! Draw black
MoveJ Offs(Target_drawing_origin,0,0,0),v100,fine,PencilHolder\WObj:=PAPER;
MoveL Offs(Target_drawing_origin,0,0,0),v50,fine,PencilHolder\WObj:=PAPER;
MoveL Offs(Target_drawing_origin,-53,0,0),v50,fine,PencilHolder\WObj:=PAPER;
MoveL Offs(Target_drawing_origin,0,1,0),v50,fine,PencilHolder\WObj:=PAPER;
MoveL Offs(Target_drawing_origin,-53,1,0),v50,fine,PencilHolder\WObj:=PAPER;
MoveL Offs(Target_drawing_origin,0,2,0),v50,fine,PencilHolder\WObj:=PAPER;
MoveL Offs(Target_drawing_origin,-53,2,0),v50,fine,PencilHolder\WObj:=PAPER;
MoveL Offs(Target_drawing_origin,0,3,0),v50,fine,PencilHolder\WObj:=PAPER;
MoveL Offs(Target_drawing_origin,-53,3,0),v50,fine,PencilHolder\WObj:=PAPER;
MoveL Offs(Target_drawing_origin,0,4,0),v50,fine,PencilHolder\WObj:=PAPER;
MoveL Offs(Target_drawing_origin,-53,4,0),v50,fine,PencilHolder\WObj:=PAPER;
MoveL Offs(Target_drawing_origin,0,5,0),v50,fine,PencilHolder\WObj:=PAPER;
MoveL Offs(Target_drawing_origin,-53,5,0),v50,fine,PencilHolder\WObj:=PAPER;
MoveL Offs(Target_drawing_origin,0,6,0),v50,fine,PencilHolder\WObj:=PAPER;
MoveL Offs(Target_drawing_origin,-58,6,0),v50,fine,PencilHolder\WObj:=PAPER;
MoveL Offs(Target_drawing_origin,0,7,0),v50,fine,PencilHolder\WObj:=PAPER;
MoveL Offs(Target_drawing_origin,-58,7,0),v50,fine,PencilHolder\WObj:=PAPER;
MoveL Offs(Target_drawing_origin,0,8,0),v50,fine,PencilHolder\WObj:=PAPER;
MoveL Offs(Target_drawing_origin,-58,8,0),v50,fine,PencilHolder\WObj:=PAPER;
MoveL Offs(Target_drawing_origin,0,9,0),v50,fine,PencilHolder\WObj:=PAPER;
MoveL Offs(Target_drawing_origin,-58,9,0),v50,fine,PencilHolder\WObj:=PAPER;
MoveL Offs(Target_drawing_origin,0,10,0),v50,fine,PencilHolder\WObj:=PAPER;
MoveL Offs(Target_drawing_origin,-58,10,0),v50,fine,PencilHolder\WObj:=PAPER;
MoveL Offs(Target_drawing_origin,0,11,0),v50,fine,PencilHolder\WObj:=PAPER;
MoveL Offs(Target_drawing_origin,-58,11,0),v50,fine,PencilHolder\WObj:=PAPER;
MoveL Offs(Target_drawing_origin,0,12,0),v50,fine,PencilHolder\WObj:=PAPER;
MoveL Offs(Target_drawing_origin,-58,12,0),v50,fine,PencilHolder\WObj:=PAPER;
MoveL Offs(Target_drawing_origin,0,13,0),v50,fine,PencilHolder\WObj:=PAPER;
MoveL Offs(Target_drawing_origin,-58,13,0),v50,fine,PencilHolder\WObj:=PAPER;
MoveL Offs(Target_drawing_origin,0,14,0),v50,fine,PencilHolder\WObj:=PAPER;
MoveL Offs(Target_drawing_origin,-58,14,0),v50,fine,PencilHolder\WObj:=PAPER;
MoveL Offs(Target_drawing_origin,0,15,0),v50,fine,PencilHolder\WObj:=PAPER;
MoveL Offs(Target_drawing_origin,-58,15,0),v50,fine,PencilHolder\WObj:=PAPER;
MoveL Offs(Target_drawing_origin,0,16,0),v50,fine,PencilHolder\WObj:=PAPER;
MoveL Offs(Target_drawing_origin,-15,16,0),v50,fine,PencilHolder\WObj:=PAPER;
MoveL Offs(Target_drawing_origin,-27,16,0),v50,fine,PencilHolder\WObj:=PAPER;
MoveL Offs(Target_drawing_origin,-58,16,0),v50,fine,PencilHolder\WObj:=PAPER;
MoveL Offs(Target_drawing_origin,0,17,0),v50,fine,PencilHolder\WObj:=PAPER;
MoveL Offs(Target_drawing_origin,-15,17,0),v50,fine,PencilHolder\WObj:=PAPER;
MoveL Offs(Target_drawing_origin,-27,17,0),v50,fine,PencilHolder\WObj:=PAPER;
MoveL Offs(Target_drawing_origin,-58,17,0),v50,fine,PencilHolder\WObj:=PAPER;
MoveL Offs(Target_drawing_origin,0,18,0),v50,fine,PencilHolder\WObj:=PAPER;
MoveL Offs(Target_drawing_origin,-15,18,0),v50,fine,PencilHolder\WObj:=PAPER;
MoveL Offs(Target_drawing_origin,-27,18,0),v50,fine,PencilHolder\WObj:=PAPER;
MoveL Offs(Target_drawing_origin,-58,18,0),v50,fine,PencilHolder\WObj:=PAPER;
MoveL Offs(Target_drawing_origin,0,19,0),v50,fine,PencilHolder\WObj:=PAPER;
MoveL Offs(Target_drawing_origin,-15,19,0),v50,fine,PencilHolder\WObj:=PAPER;
MoveL Offs(Target_drawing_origin,-27,19,0),v50,fine,PencilHolder\WObj:=PAPER;
MoveL Offs(Target_drawing_origin,-58,19,0),v50,fine,PencilHolder\WObj:=PAPER;
MoveL Offs(Target_drawing_origin,0,20,0),v50,fine,PencilHolder\WObj:=PAPER;
MoveL Offs(Target_drawing_origin,-15,20,0),v50,fine,PencilHolder\WObj:=PAPER;
MoveL Offs(Target_drawing_origin,-27,20,0),v50,fine,PencilHolder\WObj:=PAPER;
MoveL Offs(Target_drawing_origin,-58,20,0),v50,fine,PencilHolder\WObj:=PAPER;
MoveL Offs(Target_drawing_origin,-27,21,0),v50,fine,PencilHolder\WObj:=PAPER;
MoveL Offs(Target_drawing_origin,-58,21,0),v50,fine,PencilHolder\WObj:=PAPER;
MoveL Offs(Target_drawing_origin,-27,22,0),v50,fine,PencilHolder\WObj:=PAPER;
MoveL Offs(Target_drawing_origin,-58,22,0),v50,fine,PencilHolder\WObj:=PAPER;
MoveL Offs(Target_drawing_origin,-27,23,0),v50,fine,PencilHolder\WObj:=PAPER;
MoveL Offs(Target_drawing_origin,-58,23,0),v50,fine,PencilHolder\WObj:=PAPER;
MoveL Offs(Target_drawing_origin,-27,24,0),v50,fine,PencilHolder\WObj:=PAPER;
MoveL Offs(Target_drawing_origin,-58,24,0),v50,fine,PencilHolder\WObj:=PAPER;
MoveL Offs(Target_drawing_origin,-27,25,0),v50,fine,PencilHolder\WObj:=PAPER;
MoveL Offs(Target_drawing_origin,-58,25,0),v50,fine,PencilHolder\WObj:=PAPER;
MoveL Offs(Target_drawing_origin,-27,26,0),v50,fine,PencilHolder\WObj:=PAPER;
MoveL Offs(Target_drawing_origin,-58,26,0),v50,fine,PencilHolder\WObj:=PAPER;
MoveL Offs(Target_drawing_origin,-17,27,0),v50,fine,PencilHolder\WObj:=PAPER;
MoveL Offs(Target_drawing_origin,-58,27,0),v50,fine,PencilHolder\WObj:=PAPER;
MoveL Offs(Target_drawing_origin,-16,28,0),v50,fine,PencilHolder\WObj:=PAPER;
MoveL Offs(Target_drawing_origin,-58,28,0),v50,fine,PencilHolder\WObj:=PAPER;
MoveL Offs(Target_drawing_origin,-16,29,0),v50,fine,PencilHolder\WObj:=PAPER;
MoveL Offs(Target_drawing_origin,-58,29,0),v50,fine,PencilHolder\WObj:=PAPER;
MoveL Offs(Target_drawing_origin,-16,30,0),v50,fine,PencilHolder\WObj:=PAPER;
MoveL Offs(Target_drawing_origin,-58,30,0),v50,fine,PencilHolder\WObj:=PAPER;
MoveL Offs(Target_drawing_origin,-16,31,0),v50,fine,PencilHolder\WObj:=PAPER;
MoveL Offs(Target_drawing_origin,-58,31,0),v50,fine,PencilHolder\WObj:=PAPER;
MoveL Offs(Target_drawing_origin,-16,32,0),v50,fine,PencilHolder\WObj:=PAPER;
MoveL Offs(Target_drawing_origin,-58,32,0),v50,fine,PencilHolder\WObj:=PAPER;
MoveL Offs(Target_drawing_origin,-16,33,0),v50,fine,PencilHolder\WObj:=PAPER;
MoveL Offs(Target_drawing_origin,-58,33,0),v50,fine,PencilHolder\WObj:=PAPER;
MoveL Offs(Target_drawing_origin,-16,34,0),v50,fine,PencilHolder\WObj:=PAPER;
MoveL Offs(Target_drawing_origin,-58,34,0),v50,fine,PencilHolder\WObj:=PAPER;
MoveL Offs(Target_drawing_origin,-16,35,0),v50,fine,PencilHolder\WObj:=PAPER;
MoveL Offs(Target_drawing_origin,-58,35,0),v50,fine,PencilHolder\WObj:=PAPER;
MoveL Offs(Target_drawing_origin,-16,36,0),v50,fine,PencilHolder\WObj:=PAPER;
MoveL Offs(Target_drawing_origin,-58,36,0),v50,fine,PencilHolder\WObj:=PAPER;
MoveL Offs(Target_drawing_origin,-16,37,0),v50,fine,PencilHolder\WObj:=PAPER;
MoveL Offs(Target_drawing_origin,-58,37,0),v50,fine,PencilHolder\WObj:=PAPER;
MoveL Offs(Target_drawing_origin,-11,38,0),v50,fine,PencilHolder\WObj:=PAPER;
MoveL Offs(Target_drawing_origin,-53,38,0),v50,fine,PencilHolder\WObj:=PAPER;
MoveL Offs(Target_drawing_origin,-11,39,0),v50,fine,PencilHolder\WObj:=PAPER;
MoveL Offs(Target_drawing_origin,-53,39,0),v50,fine,PencilHolder\WObj:=PAPER;
MoveL Offs(Target_drawing_origin,-11,40,0),v50,fine,PencilHolder\WObj:=PAPER;
MoveL Offs(Target_drawing_origin,-53,40,0),v50,fine,PencilHolder\WObj:=PAPER;
MoveL Offs(Target_drawing_origin,-11,41,0),v50,fine,PencilHolder\WObj:=PAPER;
MoveL Offs(Target_drawing_origin,-53,41,0),v50,fine,PencilHolder\WObj:=PAPER;
MoveL Offs(Target_drawing_origin,-11,42,0),v50,fine,PencilHolder\WObj:=PAPER;
MoveL Offs(Target_drawing_origin,-53,42,0),v50,fine,PencilHolder\WObj:=PAPER;
MoveL Offs(Target_drawing_origin,-11,43,0),v50,fine,PencilHolder\WObj:=PAPER;
MoveL Offs(Target_drawing_origin,-42,43,0),v50,fine,PencilHolder\WObj:=PAPER;
MoveL Offs(Target_drawing_origin,-6,44,0),v50,fine,PencilHolder\WObj:=PAPER;
MoveL Offs(Target_drawing_origin,-42,44,0),v50,fine,PencilHolder\WObj:=PAPER;
MoveL Offs(Target_drawing_origin,-76,44,0),v50,fine,PencilHolder\WObj:=PAPER;
MoveL Offs(Target_drawing_origin,-96,44,0),v50,fine,PencilHolder\WObj:=PAPER;
MoveL Offs(Target_drawing_origin,-6,45,0),v50,fine,PencilHolder\WObj:=PAPER;
MoveL Offs(Target_drawing_origin,-42,45,0),v50,fine,PencilHolder\WObj:=PAPER;
MoveL Offs(Target_drawing_origin,-76,45,0),v50,fine,PencilHolder\WObj:=PAPER;
MoveL Offs(Target_drawing_origin,-96,45,0),v50,fine,PencilHolder\WObj:=PAPER;
MoveL Offs(Target_drawing_origin,-6,46,0),v50,fine,PencilHolder\WObj:=PAPER;
MoveL Offs(Target_drawing_origin,-42,46,0),v50,fine,PencilHolder\WObj:=PAPER;
MoveL Offs(Target_drawing_origin,-76,46,0),v50,fine,PencilHolder\WObj:=PAPER;
MoveL Offs(Target_drawing_origin,-96,46,0),v50,fine,PencilHolder\WObj:=PAPER;
MoveL Offs(Target_drawing_origin,-6,47,0),v50,fine,PencilHolder\WObj:=PAPER;
MoveL Offs(Target_drawing_origin,-42,47,0),v50,fine,PencilHolder\WObj:=PAPER;
MoveL Offs(Target_drawing_origin,-76,47,0),v50,fine,PencilHolder\WObj:=PAPER;
MoveL Offs(Target_drawing_origin,-96,47,0),v50,fine,PencilHolder\WObj:=PAPER;
MoveL Offs(Target_drawing_origin,-6,48,0),v50,fine,PencilHolder\WObj:=PAPER;
MoveL Offs(Target_drawing_origin,-37,48,0),v50,fine,PencilHolder\WObj:=PAPER;
MoveL Offs(Target_drawing_origin,-76,48,0),v50,fine,PencilHolder\WObj:=PAPER;
MoveL Offs(Target_drawing_origin,-96,48,0),v50,fine,PencilHolder\WObj:=PAPER;
MoveL Offs(Target_drawing_origin,0,49,0),v50,fine,PencilHolder\WObj:=PAPER;
MoveL Offs(Target_drawing_origin,-37,49,0),v50,fine,PencilHolder\WObj:=PAPER;
MoveL Offs(Target_drawing_origin,-71,49,0),v50,fine,PencilHolder\WObj:=PAPER;
MoveL Offs(Target_drawing_origin,-101,49,0),v50,fine,PencilHolder\WObj:=PAPER;
MoveL Offs(Target_drawing_origin,0,50,0),v50,fine,PencilHolder\WObj:=PAPER;
MoveL Offs(Target_drawing_origin,-37,50,0),v50,fine,PencilHolder\WObj:=PAPER;
MoveL Offs(Target_drawing_origin,-71,50,0),v50,fine,PencilHolder\WObj:=PAPER;
MoveL Offs(Target_drawing_origin,-101,50,0),v50,fine,PencilHolder\WObj:=PAPER;
MoveL Offs(Target_drawing_origin,0,51,0),v50,fine,PencilHolder\WObj:=PAPER;
MoveL Offs(Target_drawing_origin,-37,51,0),v50,fine,PencilHolder\WObj:=PAPER;
MoveL Offs(Target_drawing_origin,-71,51,0),v50,fine,PencilHolder\WObj:=PAPER;
MoveL Offs(Target_drawing_origin,-101,51,0),v50,fine,PencilHolder\WObj:=PAPER;
MoveL Offs(Target_drawing_origin,0,52,0),v50,fine,PencilHolder\WObj:=PAPER;
MoveL Offs(Target_drawing_origin,-37,52,0),v50,fine,PencilHolder\WObj:=PAPER;
MoveL Offs(Target_drawing_origin,-71,52,0),v50,fine,PencilHolder\WObj:=PAPER;
MoveL Offs(Target_drawing_origin,-101,52,0),v50,fine,PencilHolder\WObj:=PAPER;
MoveL Offs(Target_drawing_origin,0,53,0),v50,fine,PencilHolder\WObj:=PAPER;
MoveL Offs(Target_drawing_origin,-37,53,0),v50,fine,PencilHolder\WObj:=PAPER;
MoveL Offs(Target_drawing_origin,-71,53,0),v50,fine,PencilHolder\WObj:=PAPER;
MoveL Offs(Target_drawing_origin,-101,53,0),v50,fine,PencilHolder\WObj:=PAPER;
MoveL Offs(Target_drawing_origin,0,54,0),v50,fine,PencilHolder\WObj:=PAPER;
MoveL Offs(Target_drawing_origin,-31,54,0),v50,fine,PencilHolder\WObj:=PAPER;
MoveL Offs(Target_drawing_origin,-60,54,0),v50,fine,PencilHolder\WObj:=PAPER;
MoveL Offs(Target_drawing_origin,-107,54,0),v50,fine,PencilHolder\WObj:=PAPER;
MoveL Offs(Target_drawing_origin,0,55,0),v50,fine,PencilHolder\WObj:=PAPER;
MoveL Offs(Target_drawing_origin,-31,55,0),v50,fine,PencilHolder\WObj:=PAPER;
MoveL Offs(Target_drawing_origin,-60,55,0),v50,fine,PencilHolder\WObj:=PAPER;
MoveL Offs(Target_drawing_origin,-107,55,0),v50,fine,PencilHolder\WObj:=PAPER;
MoveL Offs(Target_drawing_origin,0,56,0),v50,fine,PencilHolder\WObj:=PAPER;
MoveL Offs(Target_drawing_origin,-31,56,0),v50,fine,PencilHolder\WObj:=PAPER;
MoveL Offs(Target_drawing_origin,-60,56,0),v50,fine,PencilHolder\WObj:=PAPER;
MoveL Offs(Target_drawing_origin,-107,56,0),v50,fine,PencilHolder\WObj:=PAPER;
MoveL Offs(Target_drawing_origin,0,57,0),v50,fine,PencilHolder\WObj:=PAPER;
MoveL Offs(Target_drawing_origin,-31,57,0),v50,fine,PencilHolder\WObj:=PAPER;
MoveL Offs(Target_drawing_origin,-60,57,0),v50,fine,PencilHolder\WObj:=PAPER;
MoveL Offs(Target_drawing_origin,-107,57,0),v50,fine,PencilHolder\WObj:=PAPER;
MoveL Offs(Target_drawing_origin,0,58,0),v50,fine,PencilHolder\WObj:=PAPER;
MoveL Offs(Target_drawing_origin,-31,58,0),v50,fine,PencilHolder\WObj:=PAPER;
MoveL Offs(Target_drawing_origin,-60,58,0),v50,fine,PencilHolder\WObj:=PAPER;
MoveL Offs(Target_drawing_origin,-107,58,0),v50,fine,PencilHolder\WObj:=PAPER;
MoveL Offs(Target_drawing_origin,0,59,0),v50,fine,PencilHolder\WObj:=PAPER;
MoveL Offs(Target_drawing_origin,-31,59,0),v50,fine,PencilHolder\WObj:=PAPER;
MoveL Offs(Target_drawing_origin,-60,59,0),v50,fine,PencilHolder\WObj:=PAPER;
MoveL Offs(Target_drawing_origin,-107,59,0),v50,fine,PencilHolder\WObj:=PAPER;
MoveL Offs(Target_drawing_origin,0,60,0),v50,fine,PencilHolder\WObj:=PAPER;
MoveL Offs(Target_drawing_origin,-112,60,0),v50,fine,PencilHolder\WObj:=PAPER;
MoveL Offs(Target_drawing_origin,0,61,0),v50,fine,PencilHolder\WObj:=PAPER;
MoveL Offs(Target_drawing_origin,-112,61,0),v50,fine,PencilHolder\WObj:=PAPER;
MoveL Offs(Target_drawing_origin,0,62,0),v50,fine,PencilHolder\WObj:=PAPER;
MoveL Offs(Target_drawing_origin,-112,62,0),v50,fine,PencilHolder\WObj:=PAPER;
MoveL Offs(Target_drawing_origin,0,63,0),v50,fine,PencilHolder\WObj:=PAPER;
MoveL Offs(Target_drawing_origin,-112,63,0),v50,fine,PencilHolder\WObj:=PAPER;
MoveL Offs(Target_drawing_origin,0,64,0),v50,fine,PencilHolder\WObj:=PAPER;
MoveL Offs(Target_drawing_origin,-112,64,0),v50,fine,PencilHolder\WObj:=PAPER;
MoveL Offs(Target_drawing_origin,0,65,0),v50,fine,PencilHolder\WObj:=PAPER;
MoveL Offs(Target_drawing_origin,-112,65,0),v50,fine,PencilHolder\WObj:=PAPER;
MoveL Offs(Target_drawing_origin,0,66,0),v50,fine,PencilHolder\WObj:=PAPER;
MoveL Offs(Target_drawing_origin,-118,66,0),v50,fine,PencilHolder\WObj:=PAPER;
MoveL Offs(Target_drawing_origin,0,67,0),v50,fine,PencilHolder\WObj:=PAPER;
MoveL Offs(Target_drawing_origin,-118,67,0),v50,fine,PencilHolder\WObj:=PAPER;
MoveL Offs(Target_drawing_origin,0,68,0),v50,fine,PencilHolder\WObj:=PAPER;
MoveL Offs(Target_drawing_origin,-118,68,0),v50,fine,PencilHolder\WObj:=PAPER;
MoveL Offs(Target_drawing_origin,0,69,0),v50,fine,PencilHolder\WObj:=PAPER;
MoveL Offs(Target_drawing_origin,-118,69,0),v50,fine,PencilHolder\WObj:=PAPER;
MoveL Offs(Target_drawing_origin,-5,70,0),v50,fine,PencilHolder\WObj:=PAPER;
MoveL Offs(Target_drawing_origin,-118,70,0),v50,fine,PencilHolder\WObj:=PAPER;
MoveL Offs(Target_drawing_origin,-6,71,0),v50,fine,PencilHolder\WObj:=PAPER;
MoveL Offs(Target_drawing_origin,-123,71,0),v50,fine,PencilHolder\WObj:=PAPER;
MoveL Offs(Target_drawing_origin,-6,72,0),v50,fine,PencilHolder\WObj:=PAPER;
MoveL Offs(Target_drawing_origin,-123,72,0),v50,fine,PencilHolder\WObj:=PAPER;
MoveL Offs(Target_drawing_origin,-6,73,0),v50,fine,PencilHolder\WObj:=PAPER;
MoveL Offs(Target_drawing_origin,-123,73,0),v50,fine,PencilHolder\WObj:=PAPER;
MoveL Offs(Target_drawing_origin,-6,74,0),v50,fine,PencilHolder\WObj:=PAPER;
MoveL Offs(Target_drawing_origin,-123,74,0),v50,fine,PencilHolder\WObj:=PAPER;
MoveL Offs(Target_drawing_origin,-6,75,0),v50,fine,PencilHolder\WObj:=PAPER;
MoveL Offs(Target_drawing_origin,-123,75,0),v50,fine,PencilHolder\WObj:=PAPER;
MoveL Offs(Target_drawing_origin,-11,76,0),v50,fine,PencilHolder\WObj:=PAPER;
MoveL Offs(Target_drawing_origin,-74,76,0),v50,fine,PencilHolder\WObj:=PAPER;
MoveL Offs(Target_drawing_origin,-92,76,0),v50,fine,PencilHolder\WObj:=PAPER;
MoveL Offs(Target_drawing_origin,-123,76,0),v50,fine,PencilHolder\WObj:=PAPER;
MoveL Offs(Target_drawing_origin,-11,77,0),v50,fine,PencilHolder\WObj:=PAPER;
MoveL Offs(Target_drawing_origin,-74,77,0),v50,fine,PencilHolder\WObj:=PAPER;
MoveL Offs(Target_drawing_origin,-92,77,0),v50,fine,PencilHolder\WObj:=PAPER;
MoveL Offs(Target_drawing_origin,-123,77,0),v50,fine,PencilHolder\WObj:=PAPER;
MoveL Offs(Target_drawing_origin,-11,78,0),v50,fine,PencilHolder\WObj:=PAPER;
MoveL Offs(Target_drawing_origin,-74,78,0),v50,fine,PencilHolder\WObj:=PAPER;
MoveL Offs(Target_drawing_origin,-92,78,0),v50,fine,PencilHolder\WObj:=PAPER;
MoveL Offs(Target_drawing_origin,-123,78,0),v50,fine,PencilHolder\WObj:=PAPER;
MoveL Offs(Target_drawing_origin,-11,79,0),v50,fine,PencilHolder\WObj:=PAPER;
MoveL Offs(Target_drawing_origin,-74,79,0),v50,fine,PencilHolder\WObj:=PAPER;
MoveL Offs(Target_drawing_origin,-92,79,0),v50,fine,PencilHolder\WObj:=PAPER;
MoveL Offs(Target_drawing_origin,-123,79,0),v50,fine,PencilHolder\WObj:=PAPER;
MoveL Offs(Target_drawing_origin,-11,80,0),v50,fine,PencilHolder\WObj:=PAPER;
MoveL Offs(Target_drawing_origin,-74,80,0),v50,fine,PencilHolder\WObj:=PAPER;
MoveL Offs(Target_drawing_origin,-92,80,0),v50,fine,PencilHolder\WObj:=PAPER;
MoveL Offs(Target_drawing_origin,-123,80,0),v50,fine,PencilHolder\WObj:=PAPER;
MoveL Offs(Target_drawing_origin,-16,81,0),v50,fine,PencilHolder\WObj:=PAPER;
MoveL Offs(Target_drawing_origin,-69,81,0),v50,fine,PencilHolder\WObj:=PAPER;
MoveL Offs(Target_drawing_origin,-92,81,0),v50,fine,PencilHolder\WObj:=PAPER;
MoveL Offs(Target_drawing_origin,-123,81,0),v50,fine,PencilHolder\WObj:=PAPER;
MoveL Offs(Target_drawing_origin,-16,82,0),v50,fine,PencilHolder\WObj:=PAPER;
MoveL Offs(Target_drawing_origin,-69,82,0),v50,fine,PencilHolder\WObj:=PAPER;
MoveL Offs(Target_drawing_origin,-92,82,0),v50,fine,PencilHolder\WObj:=PAPER;
MoveL Offs(Target_drawing_origin,-123,82,0),v50,fine,PencilHolder\WObj:=PAPER;
MoveL Offs(Target_drawing_origin,-16,83,0),v50,fine,PencilHolder\WObj:=PAPER;
MoveL Offs(Target_drawing_origin,-69,83,0),v50,fine,PencilHolder\WObj:=PAPER;
MoveL Offs(Target_drawing_origin,-92,83,0),v50,fine,PencilHolder\WObj:=PAPER;
MoveL Offs(Target_drawing_origin,-123,83,0),v50,fine,PencilHolder\WObj:=PAPER;
MoveL Offs(Target_drawing_origin,-16,84,0),v50,fine,PencilHolder\WObj:=PAPER;
MoveL Offs(Target_drawing_origin,-69,84,0),v50,fine,PencilHolder\WObj:=PAPER;
MoveL Offs(Target_drawing_origin,-92,84,0),v50,fine,PencilHolder\WObj:=PAPER;
MoveL Offs(Target_drawing_origin,-123,84,0),v50,fine,PencilHolder\WObj:=PAPER;
MoveL Offs(Target_drawing_origin,-16,85,0),v50,fine,PencilHolder\WObj:=PAPER;
MoveL Offs(Target_drawing_origin,-69,85,0),v50,fine,PencilHolder\WObj:=PAPER;
MoveL Offs(Target_drawing_origin,-92,85,0),v50,fine,PencilHolder\WObj:=PAPER;
MoveL Offs(Target_drawing_origin,-123,85,0),v50,fine,PencilHolder\WObj:=PAPER;
MoveL Offs(Target_drawing_origin,-21,86,0),v50,fine,PencilHolder\WObj:=PAPER;
MoveL Offs(Target_drawing_origin,-64,86,0),v50,fine,PencilHolder\WObj:=PAPER;
MoveL Offs(Target_drawing_origin,-92,86,0),v50,fine,PencilHolder\WObj:=PAPER;
MoveL Offs(Target_drawing_origin,-123,86,0),v50,fine,PencilHolder\WObj:=PAPER;
MoveL Offs(Target_drawing_origin,-22,87,0),v50,fine,PencilHolder\WObj:=PAPER;
MoveL Offs(Target_drawing_origin,-64,87,0),v50,fine,PencilHolder\WObj:=PAPER;
MoveL Offs(Target_drawing_origin,-87,87,0),v50,fine,PencilHolder\WObj:=PAPER;
MoveL Offs(Target_drawing_origin,-123,87,0),v50,fine,PencilHolder\WObj:=PAPER;
MoveL Offs(Target_drawing_origin,-22,88,0),v50,fine,PencilHolder\WObj:=PAPER;
MoveL Offs(Target_drawing_origin,-64,88,0),v50,fine,PencilHolder\WObj:=PAPER;
MoveL Offs(Target_drawing_origin,-87,88,0),v50,fine,PencilHolder\WObj:=PAPER;
MoveL Offs(Target_drawing_origin,-123,88,0),v50,fine,PencilHolder\WObj:=PAPER;
MoveL Offs(Target_drawing_origin,-22,89,0),v50,fine,PencilHolder\WObj:=PAPER;
MoveL Offs(Target_drawing_origin,-64,89,0),v50,fine,PencilHolder\WObj:=PAPER;
MoveL Offs(Target_drawing_origin,-87,89,0),v50,fine,PencilHolder\WObj:=PAPER;
MoveL Offs(Target_drawing_origin,-123,89,0),v50,fine,PencilHolder\WObj:=PAPER;
MoveL Offs(Target_drawing_origin,-22,90,0),v50,fine,PencilHolder\WObj:=PAPER;
MoveL Offs(Target_drawing_origin,-64,90,0),v50,fine,PencilHolder\WObj:=PAPER;
MoveL Offs(Target_drawing_origin,-87,90,0),v50,fine,PencilHolder\WObj:=PAPER;
MoveL Offs(Target_drawing_origin,-123,90,0),v50,fine,PencilHolder\WObj:=PAPER;
MoveL Offs(Target_drawing_origin,-22,91,0),v50,fine,PencilHolder\WObj:=PAPER;
MoveL Offs(Target_drawing_origin,-64,91,0),v50,fine,PencilHolder\WObj:=PAPER;
MoveL Offs(Target_drawing_origin,-87,91,0),v50,fine,PencilHolder\WObj:=PAPER;
MoveL Offs(Target_drawing_origin,-123,91,0),v50,fine,PencilHolder\WObj:=PAPER;
MoveL Offs(Target_drawing_origin,-81,92,0),v50,fine,PencilHolder\WObj:=PAPER;
MoveL Offs(Target_drawing_origin,-123,92,0),v50,fine,PencilHolder\WObj:=PAPER;
MoveL Offs(Target_drawing_origin,-81,93,0),v50,fine,PencilHolder\WObj:=PAPER;
MoveL Offs(Target_drawing_origin,-123,93,0),v50,fine,PencilHolder\WObj:=PAPER;
MoveL Offs(Target_drawing_origin,-81,94,0),v50,fine,PencilHolder\WObj:=PAPER;
MoveL Offs(Target_drawing_origin,-123,94,0),v50,fine,PencilHolder\WObj:=PAPER;
MoveL Offs(Target_drawing_origin,-81,95,0),v50,fine,PencilHolder\WObj:=PAPER;
MoveL Offs(Target_drawing_origin,-123,95,0),v50,fine,PencilHolder\WObj:=PAPER;
MoveL Offs(Target_drawing_origin,-81,96,0),v50,fine,PencilHolder\WObj:=PAPER;
MoveL Offs(Target_drawing_origin,-123,96,0),v50,fine,PencilHolder\WObj:=PAPER;
MoveL Offs(Target_drawing_origin,-81,97,0),v50,fine,PencilHolder\WObj:=PAPER;
MoveL Offs(Target_drawing_origin,-118,97,0),v50,fine,PencilHolder\WObj:=PAPER;
MoveL Offs(Target_drawing_origin,-65,98,0),v50,fine,PencilHolder\WObj:=PAPER;
MoveL Offs(Target_drawing_origin,-118,98,0),v50,fine,PencilHolder\WObj:=PAPER;
MoveL Offs(Target_drawing_origin,-65,99,0),v50,fine,PencilHolder\WObj:=PAPER;
MoveL Offs(Target_drawing_origin,-118,99,0),v50,fine,PencilHolder\WObj:=PAPER;
MoveL Offs(Target_drawing_origin,-65,100,0),v50,fine,PencilHolder\WObj:=PAPER;
MoveL Offs(Target_drawing_origin,-118,100,0),v50,fine,PencilHolder\WObj:=PAPER;
MoveL Offs(Target_drawing_origin,-65,101,0),v50,fine,PencilHolder\WObj:=PAPER;
MoveL Offs(Target_drawing_origin,-118,101,0),v50,fine,PencilHolder\WObj:=PAPER;
MoveL Offs(Target_drawing_origin,-65,102,0),v50,fine,PencilHolder\WObj:=PAPER;
MoveL Offs(Target_drawing_origin,-118,102,0),v50,fine,PencilHolder\WObj:=PAPER;
MoveL Offs(Target_drawing_origin,-49,103,0),v50,fine,PencilHolder\WObj:=PAPER;
MoveL Offs(Target_drawing_origin,-112,103,0),v50,fine,PencilHolder\WObj:=PAPER;
MoveL Offs(Target_drawing_origin,-49,104,0),v50,fine,PencilHolder\WObj:=PAPER;
MoveL Offs(Target_drawing_origin,-112,104,0),v50,fine,PencilHolder\WObj:=PAPER;
MoveL Offs(Target_drawing_origin,-49,105,0),v50,fine,PencilHolder\WObj:=PAPER;
MoveL Offs(Target_drawing_origin,-112,105,0),v50,fine,PencilHolder\WObj:=PAPER;
MoveL Offs(Target_drawing_origin,-49,106,0),v50,fine,PencilHolder\WObj:=PAPER;
MoveL Offs(Target_drawing_origin,-112,106,0),v50,fine,PencilHolder\WObj:=PAPER;
MoveL Offs(Target_drawing_origin,-49,107,0),v50,fine,PencilHolder\WObj:=PAPER;
MoveL Offs(Target_drawing_origin,-112,107,0),v50,fine,PencilHolder\WObj:=PAPER;
MoveL Offs(Target_drawing_origin,-48,108,0),v50,fine,PencilHolder\WObj:=PAPER;
MoveL Offs(Target_drawing_origin,-107,108,0),v50,fine,PencilHolder\WObj:=PAPER;
MoveL Offs(Target_drawing_origin,-44,109,0),v50,fine,PencilHolder\WObj:=PAPER;
MoveL Offs(Target_drawing_origin,-107,109,0),v50,fine,PencilHolder\WObj:=PAPER;
MoveL Offs(Target_drawing_origin,-44,110,0),v50,fine,PencilHolder\WObj:=PAPER;
MoveL Offs(Target_drawing_origin,-107,110,0),v50,fine,PencilHolder\WObj:=PAPER;
MoveL Offs(Target_drawing_origin,-44,111,0),v50,fine,PencilHolder\WObj:=PAPER;
MoveL Offs(Target_drawing_origin,-107,111,0),v50,fine,PencilHolder\WObj:=PAPER;
MoveL Offs(Target_drawing_origin,-44,112,0),v50,fine,PencilHolder\WObj:=PAPER;
MoveL Offs(Target_drawing_origin,-107,112,0),v50,fine,PencilHolder\WObj:=PAPER;
MoveL Offs(Target_drawing_origin,-43,113,0),v50,fine,PencilHolder\WObj:=PAPER;
MoveL Offs(Target_drawing_origin,-97,113,0),v50,fine,PencilHolder\WObj:=PAPER;
MoveL Offs(Target_drawing_origin,-38,114,0),v50,fine,PencilHolder\WObj:=PAPER;
MoveL Offs(Target_drawing_origin,-96,114,0),v50,fine,PencilHolder\WObj:=PAPER;
MoveL Offs(Target_drawing_origin,-38,115,0),v50,fine,PencilHolder\WObj:=PAPER;
MoveL Offs(Target_drawing_origin,-96,115,0),v50,fine,PencilHolder\WObj:=PAPER;
MoveL Offs(Target_drawing_origin,-38,116,0),v50,fine,PencilHolder\WObj:=PAPER;
MoveL Offs(Target_drawing_origin,-96,116,0),v50,fine,PencilHolder\WObj:=PAPER;
MoveL Offs(Target_drawing_origin,-38,117,0),v50,fine,PencilHolder\WObj:=PAPER;
MoveL Offs(Target_drawing_origin,-96,117,0),v50,fine,PencilHolder\WObj:=PAPER;
MoveL Offs(Target_drawing_origin,-38,118,0),v50,fine,PencilHolder\WObj:=PAPER;
MoveL Offs(Target_drawing_origin,-96,118,0),v50,fine,PencilHolder\WObj:=PAPER;
MoveL Offs(Target_drawing_origin,-38,119,0),v50,fine,PencilHolder\WObj:=PAPER;
MoveL Offs(Target_drawing_origin,-85,119,0),v50,fine,PencilHolder\WObj:=PAPER;
MoveL Offs(Target_drawing_origin,-38,120,0),v50,fine,PencilHolder\WObj:=PAPER;
MoveL Offs(Target_drawing_origin,-85,120,0),v50,fine,PencilHolder\WObj:=PAPER;
MoveL Offs(Target_drawing_origin,-38,121,0),v50,fine,PencilHolder\WObj:=PAPER;
MoveL Offs(Target_drawing_origin,-85,121,0),v50,fine,PencilHolder\WObj:=PAPER;
MoveL Offs(Target_drawing_origin,-38,122,0),v50,fine,PencilHolder\WObj:=PAPER;
MoveL Offs(Target_drawing_origin,-85,122,0),v50,fine,PencilHolder\WObj:=PAPER;
MoveL Offs(Target_drawing_origin,-38,123,0),v50,fine,PencilHolder\WObj:=PAPER;
MoveL Offs(Target_drawing_origin,-85,123,0),v50,fine,PencilHolder\WObj:=PAPER;
MoveL Offs(Target_drawing_origin,-38,124,0),v50,fine,PencilHolder\WObj:=PAPER;
MoveL Offs(Target_drawing_origin,-69,124,0),v50,fine,PencilHolder\WObj:=PAPER;
MoveL Offs(Target_drawing_origin,-33,125,0),v50,fine,PencilHolder\WObj:=PAPER;
MoveL Offs(Target_drawing_origin,-69,125,0),v50,fine,PencilHolder\WObj:=PAPER;
MoveL Offs(Target_drawing_origin,-33,126,0),v50,fine,PencilHolder\WObj:=PAPER;
MoveL Offs(Target_drawing_origin,-69,126,0),v50,fine,PencilHolder\WObj:=PAPER;
MoveL Offs(Target_drawing_origin,-33,127,0),v50,fine,PencilHolder\WObj:=PAPER;
MoveL Offs(Target_drawing_origin,-69,127,0),v50,fine,PencilHolder\WObj:=PAPER;
MoveL Offs(Target_drawing_origin,-33,128,0),v50,fine,PencilHolder\WObj:=PAPER;
MoveL Offs(Target_drawing_origin,-69,128,0),v50,fine,PencilHolder\WObj:=PAPER;
MoveL Offs(Target_drawing_origin,-33,129,0),v50,fine,PencilHolder\WObj:=PAPER;
MoveL Offs(Target_drawing_origin,-69,129,0),v50,fine,PencilHolder\WObj:=PAPER;
MoveL Offs(Target_drawing_origin,-33,130,0),v50,fine,PencilHolder\WObj:=PAPER;
MoveL Offs(Target_drawing_origin,-69,130,0),v50,fine,PencilHolder\WObj:=PAPER;
MoveL Offs(Target_drawing_origin,-27,131,0),v50,fine,PencilHolder\WObj:=PAPER;
MoveL Offs(Target_drawing_origin,-58,131,0),v50,fine,PencilHolder\WObj:=PAPER;
MoveL Offs(Target_drawing_origin,-27,132,0),v50,fine,PencilHolder\WObj:=PAPER;
MoveL Offs(Target_drawing_origin,-58,132,0),v50,fine,PencilHolder\WObj:=PAPER;
MoveL Offs(Target_drawing_origin,-27,133,0),v50,fine,PencilHolder\WObj:=PAPER;
MoveL Offs(Target_drawing_origin,-58,133,0),v50,fine,PencilHolder\WObj:=PAPER;
MoveL Offs(Target_drawing_origin,-27,134,0),v50,fine,PencilHolder\WObj:=PAPER;
MoveL Offs(Target_drawing_origin,-58,134,0),v50,fine,PencilHolder\WObj:=PAPER;
MoveL Offs(Target_drawing_origin,-27,135,0),v50,fine,PencilHolder\WObj:=PAPER;
MoveL Offs(Target_drawing_origin,-58,135,0),v50,fine,PencilHolder\WObj:=PAPER;
MoveL Offs(Target_drawing_origin,-27,136,0),v50,fine,PencilHolder\WObj:=PAPER;
MoveL Offs(Target_drawing_origin,-58,136,0),v50,fine,PencilHolder\WObj:=PAPER;
MoveL Offs(Target_drawing_origin,-27,137,0),v50,fine,PencilHolder\WObj:=PAPER;
MoveL Offs(Target_drawing_origin,-58,137,0),v50,fine,PencilHolder\WObj:=PAPER;
MoveL Offs(Target_drawing_origin,-27,138,0),v50,fine,PencilHolder\WObj:=PAPER;
MoveL Offs(Target_drawing_origin,-58,138,0),v50,fine,PencilHolder\WObj:=PAPER;
MoveL Offs(Target_drawing_origin,-27,139,0),v50,fine,PencilHolder\WObj:=PAPER;
MoveL Offs(Target_drawing_origin,-58,139,0),v50,fine,PencilHolder\WObj:=PAPER;
MoveL Offs(Target_drawing_origin,-27,140,0),v50,fine,PencilHolder\WObj:=PAPER;
MoveL Offs(Target_drawing_origin,-58,140,0),v50,fine,PencilHolder\WObj:=PAPER;
MoveL Offs(Target_drawing_origin,-27,141,0),v50,fine,PencilHolder\WObj:=PAPER;
MoveL Offs(Target_drawing_origin,-58,141,0),v50,fine,PencilHolder\WObj:=PAPER;
MoveL Offs(Target_drawing_origin,-27,142,0),v50,fine,PencilHolder\WObj:=PAPER;
MoveL Offs(Target_drawing_origin,-58,142,0),v50,fine,PencilHolder\WObj:=PAPER;
MoveL Offs(Target_drawing_origin,-27,143,0),v50,fine,PencilHolder\WObj:=PAPER;
MoveL Offs(Target_drawing_origin,-58,143,0),v50,fine,PencilHolder\WObj:=PAPER;
MoveL Offs(Target_drawing_origin,-27,144,0),v50,fine,PencilHolder\WObj:=PAPER;
MoveL Offs(Target_drawing_origin,-58,144,0),v50,fine,PencilHolder\WObj:=PAPER;
MoveL Offs(Target_drawing_origin,-27,145,0),v50,fine,PencilHolder\WObj:=PAPER;
MoveL Offs(Target_drawing_origin,-58,145,0),v50,fine,PencilHolder\WObj:=PAPER;
MoveL Offs(Target_drawing_origin,-27,146,0),v50,fine,PencilHolder\WObj:=PAPER;
MoveL Offs(Target_drawing_origin,-59,146,0),v50,fine,PencilHolder\WObj:=PAPER;
MoveL Offs(Target_drawing_origin,-27,147,0),v50,fine,PencilHolder\WObj:=PAPER;
MoveL Offs(Target_drawing_origin,-64,147,0),v50,fine,PencilHolder\WObj:=PAPER;
MoveL Offs(Target_drawing_origin,-27,148,0),v50,fine,PencilHolder\WObj:=PAPER;
MoveL Offs(Target_drawing_origin,-64,148,0),v50,fine,PencilHolder\WObj:=PAPER;
MoveL Offs(Target_drawing_origin,-27,149,0),v50,fine,PencilHolder\WObj:=PAPER;
MoveL Offs(Target_drawing_origin,-64,149,0),v50,fine,PencilHolder\WObj:=PAPER;
MoveL Offs(Target_drawing_origin,-27,150,0),v50,fine,PencilHolder\WObj:=PAPER;
MoveL Offs(Target_drawing_origin,-64,150,0),v50,fine,PencilHolder\WObj:=PAPER;
MoveL Offs(Target_drawing_origin,-27,151,0),v50,fine,PencilHolder\WObj:=PAPER;
MoveL Offs(Target_drawing_origin,-64,151,0),v50,fine,PencilHolder\WObj:=PAPER;
MoveL Offs(Target_drawing_origin,-27,152,0),v50,fine,PencilHolder\WObj:=PAPER;
MoveL Offs(Target_drawing_origin,-69,152,0),v50,fine,PencilHolder\WObj:=PAPER;
MoveL Offs(Target_drawing_origin,-108,152,0),v50,fine,PencilHolder\WObj:=PAPER;
MoveL Offs(Target_drawing_origin,-145,152,0),v50,fine,PencilHolder\WObj:=PAPER;
MoveL Offs(Target_drawing_origin,-27,153,0),v50,fine,PencilHolder\WObj:=PAPER;
MoveL Offs(Target_drawing_origin,-69,153,0),v50,fine,PencilHolder\WObj:=PAPER;
MoveL Offs(Target_drawing_origin,-108,153,0),v50,fine,PencilHolder\WObj:=PAPER;
MoveL Offs(Target_drawing_origin,-145,153,0),v50,fine,PencilHolder\WObj:=PAPER;
MoveL Offs(Target_drawing_origin,-27,154,0),v50,fine,PencilHolder\WObj:=PAPER;
MoveL Offs(Target_drawing_origin,-69,154,0),v50,fine,PencilHolder\WObj:=PAPER;
MoveL Offs(Target_drawing_origin,-108,154,0),v50,fine,PencilHolder\WObj:=PAPER;
MoveL Offs(Target_drawing_origin,-145,154,0),v50,fine,PencilHolder\WObj:=PAPER;
MoveL Offs(Target_drawing_origin,-27,155,0),v50,fine,PencilHolder\WObj:=PAPER;
MoveL Offs(Target_drawing_origin,-69,155,0),v50,fine,PencilHolder\WObj:=PAPER;
MoveL Offs(Target_drawing_origin,-108,155,0),v50,fine,PencilHolder\WObj:=PAPER;
MoveL Offs(Target_drawing_origin,-145,155,0),v50,fine,PencilHolder\WObj:=PAPER;
MoveL Offs(Target_drawing_origin,-27,156,0),v50,fine,PencilHolder\WObj:=PAPER;
MoveL Offs(Target_drawing_origin,-69,156,0),v50,fine,PencilHolder\WObj:=PAPER;
MoveL Offs(Target_drawing_origin,-108,156,0),v50,fine,PencilHolder\WObj:=PAPER;
MoveL Offs(Target_drawing_origin,-145,156,0),v50,fine,PencilHolder\WObj:=PAPER;
MoveL Offs(Target_drawing_origin,-33,157,0),v50,fine,PencilHolder\WObj:=PAPER;
MoveL Offs(Target_drawing_origin,-150,157,0),v50,fine,PencilHolder\WObj:=PAPER;
MoveL Offs(Target_drawing_origin,-33,158,0),v50,fine,PencilHolder\WObj:=PAPER;
MoveL Offs(Target_drawing_origin,-150,158,0),v50,fine,PencilHolder\WObj:=PAPER;
MoveL Offs(Target_drawing_origin,-33,159,0),v50,fine,PencilHolder\WObj:=PAPER;
MoveL Offs(Target_drawing_origin,-150,159,0),v50,fine,PencilHolder\WObj:=PAPER;
MoveL Offs(Target_drawing_origin,-33,160,0),v50,fine,PencilHolder\WObj:=PAPER;
MoveL Offs(Target_drawing_origin,-150,160,0),v50,fine,PencilHolder\WObj:=PAPER;
MoveL Offs(Target_drawing_origin,-33,161,0),v50,fine,PencilHolder\WObj:=PAPER;
MoveL Offs(Target_drawing_origin,-150,161,0),v50,fine,PencilHolder\WObj:=PAPER;
MoveL Offs(Target_drawing_origin,-38,162,0),v50,fine,PencilHolder\WObj:=PAPER;
MoveL Offs(Target_drawing_origin,-150,162,0),v50,fine,PencilHolder\WObj:=PAPER;
MoveL Offs(Target_drawing_origin,-38,163,0),v50,fine,PencilHolder\WObj:=PAPER;
MoveL Offs(Target_drawing_origin,-156,163,0),v50,fine,PencilHolder\WObj:=PAPER;
MoveL Offs(Target_drawing_origin,-38,164,0),v50,fine,PencilHolder\WObj:=PAPER;
MoveL Offs(Target_drawing_origin,-156,164,0),v50,fine,PencilHolder\WObj:=PAPER;
MoveL Offs(Target_drawing_origin,-38,165,0),v50,fine,PencilHolder\WObj:=PAPER;
MoveL Offs(Target_drawing_origin,-156,165,0),v50,fine,PencilHolder\WObj:=PAPER;
MoveL Offs(Target_drawing_origin,-38,166,0),v50,fine,PencilHolder\WObj:=PAPER;
MoveL Offs(Target_drawing_origin,-156,166,0),v50,fine,PencilHolder\WObj:=PAPER;
MoveL Offs(Target_drawing_origin,-38,167,0),v50,fine,PencilHolder\WObj:=PAPER;
MoveL Offs(Target_drawing_origin,-156,167,0),v50,fine,PencilHolder\WObj:=PAPER;
MoveL Offs(Target_drawing_origin,-44,168,0),v50,fine,PencilHolder\WObj:=PAPER;
MoveL Offs(Target_drawing_origin,-156,168,0),v50,fine,PencilHolder\WObj:=PAPER;
MoveL Offs(Target_drawing_origin,-44,169,0),v50,fine,PencilHolder\WObj:=PAPER;
MoveL Offs(Target_drawing_origin,-156,169,0),v50,fine,PencilHolder\WObj:=PAPER;
MoveL Offs(Target_drawing_origin,-44,170,0),v50,fine,PencilHolder\WObj:=PAPER;
MoveL Offs(Target_drawing_origin,-156,170,0),v50,fine,PencilHolder\WObj:=PAPER;
MoveL Offs(Target_drawing_origin,-44,171,0),v50,fine,PencilHolder\WObj:=PAPER;
MoveL Offs(Target_drawing_origin,-156,171,0),v50,fine,PencilHolder\WObj:=PAPER;
MoveL Offs(Target_drawing_origin,-44,172,0),v50,fine,PencilHolder\WObj:=PAPER;
MoveL Offs(Target_drawing_origin,-156,172,0),v50,fine,PencilHolder\WObj:=PAPER;
MoveL Offs(Target_drawing_origin,-54,173,0),v50,fine,PencilHolder\WObj:=PAPER;
MoveL Offs(Target_drawing_origin,-123,173,0),v50,fine,PencilHolder\WObj:=PAPER;
MoveL Offs(Target_drawing_origin,-130,173,0),v50,fine,PencilHolder\WObj:=PAPER;
MoveL Offs(Target_drawing_origin,-156,173,0),v50,fine,PencilHolder\WObj:=PAPER;
MoveL Offs(Target_drawing_origin,-54,174,0),v50,fine,PencilHolder\WObj:=PAPER;
MoveL Offs(Target_drawing_origin,-123,174,0),v50,fine,PencilHolder\WObj:=PAPER;
MoveL Offs(Target_drawing_origin,-130,174,0),v50,fine,PencilHolder\WObj:=PAPER;
MoveL Offs(Target_drawing_origin,-156,174,0),v50,fine,PencilHolder\WObj:=PAPER;
MoveL Offs(Target_drawing_origin,-54,175,0),v50,fine,PencilHolder\WObj:=PAPER;
MoveL Offs(Target_drawing_origin,-123,175,0),v50,fine,PencilHolder\WObj:=PAPER;
MoveL Offs(Target_drawing_origin,-130,175,0),v50,fine,PencilHolder\WObj:=PAPER;
MoveL Offs(Target_drawing_origin,-156,175,0),v50,fine,PencilHolder\WObj:=PAPER;
MoveL Offs(Target_drawing_origin,-54,176,0),v50,fine,PencilHolder\WObj:=PAPER;
MoveL Offs(Target_drawing_origin,-123,176,0),v50,fine,PencilHolder\WObj:=PAPER;
MoveL Offs(Target_drawing_origin,-130,176,0),v50,fine,PencilHolder\WObj:=PAPER;
MoveL Offs(Target_drawing_origin,-156,176,0),v50,fine,PencilHolder\WObj:=PAPER;
MoveL Offs(Target_drawing_origin,-54,177,0),v50,fine,PencilHolder\WObj:=PAPER;
MoveL Offs(Target_drawing_origin,-123,177,0),v50,fine,PencilHolder\WObj:=PAPER;
MoveL Offs(Target_drawing_origin,-130,177,0),v50,fine,PencilHolder\WObj:=PAPER;
MoveL Offs(Target_drawing_origin,-156,177,0),v50,fine,PencilHolder\WObj:=PAPER;
MoveL Offs(Target_drawing_origin,-59,178,0),v50,fine,PencilHolder\WObj:=PAPER;
MoveL Offs(Target_drawing_origin,-118,178,0),v50,fine,PencilHolder\WObj:=PAPER;
MoveL Offs(Target_drawing_origin,-130,178,0),v50,fine,PencilHolder\WObj:=PAPER;
MoveL Offs(Target_drawing_origin,-156,178,0),v50,fine,PencilHolder\WObj:=PAPER;
MoveL Offs(Target_drawing_origin,-60,179,0),v50,fine,PencilHolder\WObj:=PAPER;
MoveL Offs(Target_drawing_origin,-118,179,0),v50,fine,PencilHolder\WObj:=PAPER;
MoveL Offs(Target_drawing_origin,-130,179,0),v50,fine,PencilHolder\WObj:=PAPER;
MoveL Offs(Target_drawing_origin,-156,179,0),v50,fine,PencilHolder\WObj:=PAPER;
MoveL Offs(Target_drawing_origin,-60,180,0),v50,fine,PencilHolder\WObj:=PAPER;
MoveL Offs(Target_drawing_origin,-118,180,0),v50,fine,PencilHolder\WObj:=PAPER;
MoveL Offs(Target_drawing_origin,-130,180,0),v50,fine,PencilHolder\WObj:=PAPER;
MoveL Offs(Target_drawing_origin,-156,180,0),v50,fine,PencilHolder\WObj:=PAPER;
MoveL Offs(Target_drawing_origin,-60,181,0),v50,fine,PencilHolder\WObj:=PAPER;
MoveL Offs(Target_drawing_origin,-118,181,0),v50,fine,PencilHolder\WObj:=PAPER;
MoveL Offs(Target_drawing_origin,-130,181,0),v50,fine,PencilHolder\WObj:=PAPER;
MoveL Offs(Target_drawing_origin,-156,181,0),v50,fine,PencilHolder\WObj:=PAPER;
MoveL Offs(Target_drawing_origin,-60,182,0),v50,fine,PencilHolder\WObj:=PAPER;
MoveL Offs(Target_drawing_origin,-118,182,0),v50,fine,PencilHolder\WObj:=PAPER;
MoveL Offs(Target_drawing_origin,-130,182,0),v50,fine,PencilHolder\WObj:=PAPER;
MoveL Offs(Target_drawing_origin,-156,182,0),v50,fine,PencilHolder\WObj:=PAPER;
MoveL Offs(Target_drawing_origin,-60,183,0),v50,fine,PencilHolder\WObj:=PAPER;
MoveL Offs(Target_drawing_origin,-118,183,0),v50,fine,PencilHolder\WObj:=PAPER;
MoveL Offs(Target_drawing_origin,-130,183,0),v50,fine,PencilHolder\WObj:=PAPER;
MoveL Offs(Target_drawing_origin,-156,183,0),v50,fine,PencilHolder\WObj:=PAPER;
MoveL Offs(Target_drawing_origin,-119,184,0),v50,fine,PencilHolder\WObj:=PAPER;
MoveL Offs(Target_drawing_origin,-156,184,0),v50,fine,PencilHolder\WObj:=PAPER;
MoveL Offs(Target_drawing_origin,-119,185,0),v50,fine,PencilHolder\WObj:=PAPER;
MoveL Offs(Target_drawing_origin,-156,185,0),v50,fine,PencilHolder\WObj:=PAPER;
MoveL Offs(Target_drawing_origin,-119,186,0),v50,fine,PencilHolder\WObj:=PAPER;
MoveL Offs(Target_drawing_origin,-156,186,0),v50,fine,PencilHolder\WObj:=PAPER;
MoveL Offs(Target_drawing_origin,-119,187,0),v50,fine,PencilHolder\WObj:=PAPER;
MoveL Offs(Target_drawing_origin,-156,187,0),v50,fine,PencilHolder\WObj:=PAPER;
MoveL Offs(Target_drawing_origin,-119,188,0),v50,fine,PencilHolder\WObj:=PAPER;
MoveL Offs(Target_drawing_origin,-156,188,0),v50,fine,PencilHolder\WObj:=PAPER;
MoveL Offs(Target_drawing_origin,-119,189,0),v50,fine,PencilHolder\WObj:=PAPER;
MoveL Offs(Target_drawing_origin,-156,189,0),v50,fine,PencilHolder\WObj:=PAPER;
MoveL Offs(Target_drawing_origin,-44,190,0),v50,fine,PencilHolder\WObj:=PAPER;
MoveL Offs(Target_drawing_origin,-85,190,0),v50,fine,PencilHolder\WObj:=PAPER;
MoveL Offs(Target_drawing_origin,-103,190,0),v50,fine,PencilHolder\WObj:=PAPER;
MoveL Offs(Target_drawing_origin,-156,190,0),v50,fine,PencilHolder\WObj:=PAPER;
MoveL Offs(Target_drawing_origin,-44,191,0),v50,fine,PencilHolder\WObj:=PAPER;
MoveL Offs(Target_drawing_origin,-85,191,0),v50,fine,PencilHolder\WObj:=PAPER;
MoveL Offs(Target_drawing_origin,-103,191,0),v50,fine,PencilHolder\WObj:=PAPER;
MoveL Offs(Target_drawing_origin,-156,191,0),v50,fine,PencilHolder\WObj:=PAPER;
MoveL Offs(Target_drawing_origin,-44,192,0),v50,fine,PencilHolder\WObj:=PAPER;
MoveL Offs(Target_drawing_origin,-85,192,0),v50,fine,PencilHolder\WObj:=PAPER;
MoveL Offs(Target_drawing_origin,-103,192,0),v50,fine,PencilHolder\WObj:=PAPER;
MoveL Offs(Target_drawing_origin,-156,192,0),v50,fine,PencilHolder\WObj:=PAPER;
MoveL Offs(Target_drawing_origin,-44,193,0),v50,fine,PencilHolder\WObj:=PAPER;
MoveL Offs(Target_drawing_origin,-85,193,0),v50,fine,PencilHolder\WObj:=PAPER;
MoveL Offs(Target_drawing_origin,-103,193,0),v50,fine,PencilHolder\WObj:=PAPER;
MoveL Offs(Target_drawing_origin,-156,193,0),v50,fine,PencilHolder\WObj:=PAPER;
MoveL Offs(Target_drawing_origin,-44,194,0),v50,fine,PencilHolder\WObj:=PAPER;
MoveL Offs(Target_drawing_origin,-85,194,0),v50,fine,PencilHolder\WObj:=PAPER;
MoveL Offs(Target_drawing_origin,-103,194,0),v50,fine,PencilHolder\WObj:=PAPER;
MoveL Offs(Target_drawing_origin,-156,194,0),v50,fine,PencilHolder\WObj:=PAPER;
MoveL Offs(Target_drawing_origin,-33,195,0),v50,fine,PencilHolder\WObj:=PAPER;
MoveL Offs(Target_drawing_origin,-150,195,0),v50,fine,PencilHolder\WObj:=PAPER;
MoveL Offs(Target_drawing_origin,-33,196,0),v50,fine,PencilHolder\WObj:=PAPER;
MoveL Offs(Target_drawing_origin,-150,196,0),v50,fine,PencilHolder\WObj:=PAPER;
MoveL Offs(Target_drawing_origin,-33,197,0),v50,fine,PencilHolder\WObj:=PAPER;
MoveL Offs(Target_drawing_origin,-150,197,0),v50,fine,PencilHolder\WObj:=PAPER;
MoveL Offs(Target_drawing_origin,-33,198,0),v50,fine,PencilHolder\WObj:=PAPER;
MoveL Offs(Target_drawing_origin,-150,198,0),v50,fine,PencilHolder\WObj:=PAPER;
MoveL Offs(Target_drawing_origin,-33,199,0),v50,fine,PencilHolder\WObj:=PAPER;
MoveL Offs(Target_drawing_origin,-150,199,0),v50,fine,PencilHolder\WObj:=PAPER;
MoveL Offs(Target_drawing_origin,-32,200,0),v50,fine,PencilHolder\WObj:=PAPER;
MoveL Offs(Target_drawing_origin,-145,200,0),v50,fine,PencilHolder\WObj:=PAPER;
MoveL Offs(Target_drawing_origin,-27,201,0),v50,fine,PencilHolder\WObj:=PAPER;
MoveL Offs(Target_drawing_origin,-145,201,0),v50,fine,PencilHolder\WObj:=PAPER;
MoveL Offs(Target_drawing_origin,-27,202,0),v50,fine,PencilHolder\WObj:=PAPER;
MoveL Offs(Target_drawing_origin,-145,202,0),v50,fine,PencilHolder\WObj:=PAPER;
MoveL Offs(Target_drawing_origin,-27,203,0),v50,fine,PencilHolder\WObj:=PAPER;
MoveL Offs(Target_drawing_origin,-145,203,0),v50,fine,PencilHolder\WObj:=PAPER;
MoveL Offs(Target_drawing_origin,-27,204,0),v50,fine,PencilHolder\WObj:=PAPER;
MoveL Offs(Target_drawing_origin,-145,204,0),v50,fine,PencilHolder\WObj:=PAPER;
MoveL Offs(Target_drawing_origin,-27,205,0),v50,fine,PencilHolder\WObj:=PAPER;
MoveL Offs(Target_drawing_origin,-145,205,0),v50,fine,PencilHolder\WObj:=PAPER;
MoveL Offs(Target_drawing_origin,-22,206,0),v50,fine,PencilHolder\WObj:=PAPER;
MoveL Offs(Target_drawing_origin,-139,206,0),v50,fine,PencilHolder\WObj:=PAPER;
MoveL Offs(Target_drawing_origin,-22,207,0),v50,fine,PencilHolder\WObj:=PAPER;
MoveL Offs(Target_drawing_origin,-139,207,0),v50,fine,PencilHolder\WObj:=PAPER;
MoveL Offs(Target_drawing_origin,-22,208,0),v50,fine,PencilHolder\WObj:=PAPER;
MoveL Offs(Target_drawing_origin,-139,208,0),v50,fine,PencilHolder\WObj:=PAPER;
MoveL Offs(Target_drawing_origin,-22,209,0),v50,fine,PencilHolder\WObj:=PAPER;
MoveL Offs(Target_drawing_origin,-139,209,0),v50,fine,PencilHolder\WObj:=PAPER;
MoveL Offs(Target_drawing_origin,-22,210,0),v50,fine,PencilHolder\WObj:=PAPER;
MoveL Offs(Target_drawing_origin,-139,210,0),v50,fine,PencilHolder\WObj:=PAPER;
MoveL Offs(Target_drawing_origin,-21,211,0),v50,fine,PencilHolder\WObj:=PAPER;
MoveL Offs(Target_drawing_origin,-64,211,0),v50,fine,PencilHolder\WObj:=PAPER;
MoveL Offs(Target_drawing_origin,-70,211,0),v50,fine,PencilHolder\WObj:=PAPER;
MoveL Offs(Target_drawing_origin,-123,211,0),v50,fine,PencilHolder\WObj:=PAPER;
MoveL Offs(Target_drawing_origin,-16,212,0),v50,fine,PencilHolder\WObj:=PAPER;
MoveL Offs(Target_drawing_origin,-64,212,0),v50,fine,PencilHolder\WObj:=PAPER;
MoveL Offs(Target_drawing_origin,-71,212,0),v50,fine,PencilHolder\WObj:=PAPER;
MoveL Offs(Target_drawing_origin,-123,212,0),v50,fine,PencilHolder\WObj:=PAPER;
MoveL Offs(Target_drawing_origin,-16,213,0),v50,fine,PencilHolder\WObj:=PAPER;
MoveL Offs(Target_drawing_origin,-64,213,0),v50,fine,PencilHolder\WObj:=PAPER;
MoveL Offs(Target_drawing_origin,-71,213,0),v50,fine,PencilHolder\WObj:=PAPER;
MoveL Offs(Target_drawing_origin,-123,213,0),v50,fine,PencilHolder\WObj:=PAPER;
MoveL Offs(Target_drawing_origin,-16,214,0),v50,fine,PencilHolder\WObj:=PAPER;
MoveL Offs(Target_drawing_origin,-64,214,0),v50,fine,PencilHolder\WObj:=PAPER;
MoveL Offs(Target_drawing_origin,-71,214,0),v50,fine,PencilHolder\WObj:=PAPER;
MoveL Offs(Target_drawing_origin,-123,214,0),v50,fine,PencilHolder\WObj:=PAPER;
MoveL Offs(Target_drawing_origin,-16,215,0),v50,fine,PencilHolder\WObj:=PAPER;
MoveL Offs(Target_drawing_origin,-64,215,0),v50,fine,PencilHolder\WObj:=PAPER;
MoveL Offs(Target_drawing_origin,-71,215,0),v50,fine,PencilHolder\WObj:=PAPER;
MoveL Offs(Target_drawing_origin,-123,215,0),v50,fine,PencilHolder\WObj:=PAPER;
MoveL Offs(Target_drawing_origin,-16,216,0),v50,fine,PencilHolder\WObj:=PAPER;
MoveL Offs(Target_drawing_origin,-48,216,0),v50,fine,PencilHolder\WObj:=PAPER;
MoveL Offs(Target_drawing_origin,-16,217,0),v50,fine,PencilHolder\WObj:=PAPER;
MoveL Offs(Target_drawing_origin,-47,217,0),v50,fine,PencilHolder\WObj:=PAPER;
MoveL Offs(Target_drawing_origin,-16,218,0),v50,fine,PencilHolder\WObj:=PAPER;
MoveL Offs(Target_drawing_origin,-47,218,0),v50,fine,PencilHolder\WObj:=PAPER;
MoveL Offs(Target_drawing_origin,-16,219,0),v50,fine,PencilHolder\WObj:=PAPER;
MoveL Offs(Target_drawing_origin,-47,219,0),v50,fine,PencilHolder\WObj:=PAPER;
MoveL Offs(Target_drawing_origin,-16,220,0),v50,fine,PencilHolder\WObj:=PAPER;
MoveL Offs(Target_drawing_origin,-47,220,0),v50,fine,PencilHolder\WObj:=PAPER;
MoveL Offs(Target_drawing_origin,-16,221,0),v50,fine,PencilHolder\WObj:=PAPER;
MoveL Offs(Target_drawing_origin,-47,221,0),v50,fine,PencilHolder\WObj:=PAPER;
MoveL Offs(Target_drawing_origin,-16,222,0),v50,fine,PencilHolder\WObj:=PAPER;
MoveL Offs(Target_drawing_origin,-69,222,0),v50,fine,PencilHolder\WObj:=PAPER;
MoveL Offs(Target_drawing_origin,-16,223,0),v50,fine,PencilHolder\WObj:=PAPER;
MoveL Offs(Target_drawing_origin,-69,223,0),v50,fine,PencilHolder\WObj:=PAPER;
MoveL Offs(Target_drawing_origin,-16,224,0),v50,fine,PencilHolder\WObj:=PAPER;
MoveL Offs(Target_drawing_origin,-69,224,0),v50,fine,PencilHolder\WObj:=PAPER;
MoveL Offs(Target_drawing_origin,-16,225,0),v50,fine,PencilHolder\WObj:=PAPER;
MoveL Offs(Target_drawing_origin,-69,225,0),v50,fine,PencilHolder\WObj:=PAPER;
MoveL Offs(Target_drawing_origin,-16,226,0),v50,fine,PencilHolder\WObj:=PAPER;
MoveL Offs(Target_drawing_origin,-69,226,0),v50,fine,PencilHolder\WObj:=PAPER;
MoveL Offs(Target_drawing_origin,-16,227,0),v50,fine,PencilHolder\WObj:=PAPER;
MoveL Offs(Target_drawing_origin,-69,227,0),v50,fine,PencilHolder\WObj:=PAPER;
MoveL Offs(Target_drawing_origin,-16,228,0),v50,fine,PencilHolder\WObj:=PAPER;
MoveL Offs(Target_drawing_origin,-139,228,0),v50,fine,PencilHolder\WObj:=PAPER;
MoveL Offs(Target_drawing_origin,-16,229,0),v50,fine,PencilHolder\WObj:=PAPER;
MoveL Offs(Target_drawing_origin,-139,229,0),v50,fine,PencilHolder\WObj:=PAPER;
MoveL Offs(Target_drawing_origin,-16,230,0),v50,fine,PencilHolder\WObj:=PAPER;
MoveL Offs(Target_drawing_origin,-139,230,0),v50,fine,PencilHolder\WObj:=PAPER;
MoveL Offs(Target_drawing_origin,-16,231,0),v50,fine,PencilHolder\WObj:=PAPER;
MoveL Offs(Target_drawing_origin,-139,231,0),v50,fine,PencilHolder\WObj:=PAPER;
MoveL Offs(Target_drawing_origin,-17,232,0),v50,fine,PencilHolder\WObj:=PAPER;
MoveL Offs(Target_drawing_origin,-139,232,0),v50,fine,PencilHolder\WObj:=PAPER;
MoveL Offs(Target_drawing_origin,-22,233,0),v50,fine,PencilHolder\WObj:=PAPER;
MoveL Offs(Target_drawing_origin,-161,233,0),v50,fine,PencilHolder\WObj:=PAPER;
MoveL Offs(Target_drawing_origin,-22,234,0),v50,fine,PencilHolder\WObj:=PAPER;
MoveL Offs(Target_drawing_origin,-161,234,0),v50,fine,PencilHolder\WObj:=PAPER;
MoveL Offs(Target_drawing_origin,-22,235,0),v50,fine,PencilHolder\WObj:=PAPER;
MoveL Offs(Target_drawing_origin,-161,235,0),v50,fine,PencilHolder\WObj:=PAPER;
MoveL Offs(Target_drawing_origin,-22,236,0),v50,fine,PencilHolder\WObj:=PAPER;
MoveL Offs(Target_drawing_origin,-161,236,0),v50,fine,PencilHolder\WObj:=PAPER;
MoveL Offs(Target_drawing_origin,-22,237,0),v50,fine,PencilHolder\WObj:=PAPER;
MoveL Offs(Target_drawing_origin,-161,237,0),v50,fine,PencilHolder\WObj:=PAPER;
MoveL Offs(Target_drawing_origin,-27,238,0),v50,fine,PencilHolder\WObj:=PAPER;
MoveL Offs(Target_drawing_origin,-161,238,0),v50,fine,PencilHolder\WObj:=PAPER;
MoveL Offs(Target_drawing_origin,-27,239,0),v50,fine,PencilHolder\WObj:=PAPER;
MoveL Offs(Target_drawing_origin,-172,239,0),v50,fine,PencilHolder\WObj:=PAPER;
MoveL Offs(Target_drawing_origin,-27,240,0),v50,fine,PencilHolder\WObj:=PAPER;
MoveL Offs(Target_drawing_origin,-172,240,0),v50,fine,PencilHolder\WObj:=PAPER;
MoveL Offs(Target_drawing_origin,-27,241,0),v50,fine,PencilHolder\WObj:=PAPER;
MoveL Offs(Target_drawing_origin,-172,241,0),v50,fine,PencilHolder\WObj:=PAPER;
MoveL Offs(Target_drawing_origin,-27,242,0),v50,fine,PencilHolder\WObj:=PAPER;
MoveL Offs(Target_drawing_origin,-172,242,0),v50,fine,PencilHolder\WObj:=PAPER;
MoveL Offs(Target_drawing_origin,-54,243,0),v50,fine,PencilHolder\WObj:=PAPER;
MoveL Offs(Target_drawing_origin,-172,243,0),v50,fine,PencilHolder\WObj:=PAPER;
MoveL Offs(Target_drawing_origin,-54,244,0),v50,fine,PencilHolder\WObj:=PAPER;
MoveL Offs(Target_drawing_origin,-172,244,0),v50,fine,PencilHolder\WObj:=PAPER;
MoveL Offs(Target_drawing_origin,-54,245,0),v50,fine,PencilHolder\WObj:=PAPER;
MoveL Offs(Target_drawing_origin,-172,245,0),v50,fine,PencilHolder\WObj:=PAPER;
MoveL Offs(Target_drawing_origin,-54,246,0),v50,fine,PencilHolder\WObj:=PAPER;
MoveL Offs(Target_drawing_origin,-172,246,0),v50,fine,PencilHolder\WObj:=PAPER;
MoveL Offs(Target_drawing_origin,-54,247,0),v50,fine,PencilHolder\WObj:=PAPER;
MoveL Offs(Target_drawing_origin,-172,247,0),v50,fine,PencilHolder\WObj:=PAPER;
MoveL Offs(Target_drawing_origin,-54,248,0),v50,fine,PencilHolder\WObj:=PAPER;
MoveL Offs(Target_drawing_origin,-172,248,0),v50,fine,PencilHolder\WObj:=PAPER;
MoveL Offs(Target_drawing_origin,-125,249,0),v50,fine,PencilHolder\WObj:=PAPER;
MoveL Offs(Target_drawing_origin,-172,249,0),v50,fine,PencilHolder\WObj:=PAPER;
MoveL Offs(Target_drawing_origin,-125,250,0),v50,fine,PencilHolder\WObj:=PAPER;
MoveL Offs(Target_drawing_origin,-172,250,0),v50,fine,PencilHolder\WObj:=PAPER;
MoveL Offs(Target_drawing_origin,-125,251,0),v50,fine,PencilHolder\WObj:=PAPER;
MoveL Offs(Target_drawing_origin,-172,251,0),v50,fine,PencilHolder\WObj:=PAPER;
MoveL Offs(Target_drawing_origin,-125,252,0),v50,fine,PencilHolder\WObj:=PAPER;
MoveL Offs(Target_drawing_origin,-172,252,0),v50,fine,PencilHolder\WObj:=PAPER;
MoveL Offs(Target_drawing_origin,-125,253,0),v50,fine,PencilHolder\WObj:=PAPER;
MoveL Offs(Target_drawing_origin,-172,253,0),v50,fine,PencilHolder\WObj:=PAPER;
MoveL Offs(Target_drawing_origin,-146,254,0),v50,fine,PencilHolder\WObj:=PAPER;
MoveL Offs(Target_drawing_origin,-172,254,0),v50,fine,PencilHolder\WObj:=PAPER;
MoveL Offs(Target_drawing_origin,-146,255,0),v50,fine,PencilHolder\WObj:=PAPER;
MoveL Offs(Target_drawing_origin,-172,255,0),v50,fine,PencilHolder\WObj:=PAPER;
MoveL Offs(Target_drawing_origin,-146,256,0),v50,fine,PencilHolder\WObj:=PAPER;
MoveL Offs(Target_drawing_origin,-172,256,0),v50,fine,PencilHolder\WObj:=PAPER;
MoveL Offs(Target_drawing_origin,-146,257,0),v50,fine,PencilHolder\WObj:=PAPER;
MoveL Offs(Target_drawing_origin,-172,257,0),v50,fine,PencilHolder\WObj:=PAPER;
MoveL Offs(Target_drawing_origin,-146,258,0),v50,fine,PencilHolder\WObj:=PAPER;
MoveL Offs(Target_drawing_origin,-172,258,0),v50,fine,PencilHolder\WObj:=PAPER;
MoveL Offs(Target_drawing_origin,-146,259,0),v50,fine,PencilHolder\WObj:=PAPER;
MoveL Offs(Target_drawing_origin,-172,259,0),v50,fine,PencilHolder\WObj:=PAPER;


ENDPROC


ENDMODULE
